// TIA Portal V19 export
VAR_GLOBAL   // PLC tag table "TT - Plate"
   iPlateSenCilPushingIn_d0 AT %I1.0 : Bool;   // Terugkoppeling pusher roteren plaat
   iPlateSenInductive_dm AT %I1.6 : Bool;   // True when metallic
   iPlateSenPresence_dp AT %I1.7 : Bool;
   iPlateSenNotBlack AT %I2.0 : Bool;   // Niet definitief, True when nothing and white
   "oPlateVenCilPushing_D+" AT %Q0.4 : Bool;
   "oPlateVenCilLocking_E+" AT %Q0.5 : Bool;
   "oPlateVenCilMeasuringDown_L+" AT %Q1.6 : Bool;
   iPlateSenHeight AT %IW65 : Int;
END_VAR
